PROGRAM MAIN
VAR
	

END_VAR

END_PROGRAM

(* stored: Version 1.1.0.1, ProductVersion 3.1.4022.12
   POU MAIN: Id {61478f02-8d40-4f8a-8139-c326911315d5}, SpecialFunc None *)
